// TIA Portal project "Practica_7_V14" (V14)
// Primer proyecto - practica experimental 7

(* hardware
DEVICE "S7-1200 station_1"  S7-1200 Station
   slot 0: "Rack_0"  Rack  V1.0
   slot 1: "PLC_1"  CPU 1214C DC/DC/DC  6ES7 214-1AG40-0XB0  V4.2
*)

// ===== PLC "PLC_1"  CPU 1214C DC/DC/DC =====

VAR_GLOBAL   // PLC tag table "Default tag table"
   "PM" AT %I0.0 : Bool;
   "PP" AT %I0.1 : Bool;
   "MOTOR" AT %Q0.0 : Bool;
   "APAGADO" AT %M0.1 : Bool;
   "ENCENDIDO" AT %M0.0 : Bool;
   "IL" AT %Q0.1 : Bool;
   "DP" AT %I0.2 : Bool;
   "CU" AT %M0.3 : Bool;
   "MEMORIA_RESET_CNT" AT %M0.2 : Bool;
END_VAR

// folder: System blocks/Program resources

DATA_BLOCK "CNT_UP"   // DB1
{ S7_Optimized_Access := 'TRUE' }
AUTHOR : Simatic
FAMILY : IEC
NAME : CNTR
VERSION : 1.0
// stored: InstanceOfName IEC_COUNTER
"IEC_COUNTER"
BEGIN
END_DATA_BLOCK

// folder: (top level)

ORGANIZATION_BLOCK "Main"   // OB1, LAD, ProgramCycle
TITLE = "Main Program Sweep (Cycle)"
{ S7_Optimized_Access := 'TRUE' }
VERSION : 0.1
   VAR_INPUT
      Initial_Call : Bool;   // Initial call of this OB
      Remanence : Bool;   // =True, if remanent data are available
   END_VAR
   VAR CONSTANT
      MAX_CNT : Int := 4;
   END_VAR
   VAR_TEMP   // added for the SCL form of the ladder/FBD networks
      _w1 : Bool;
   END_VAR
BEGIN

REGION Network 1
   // INICIALIZACION
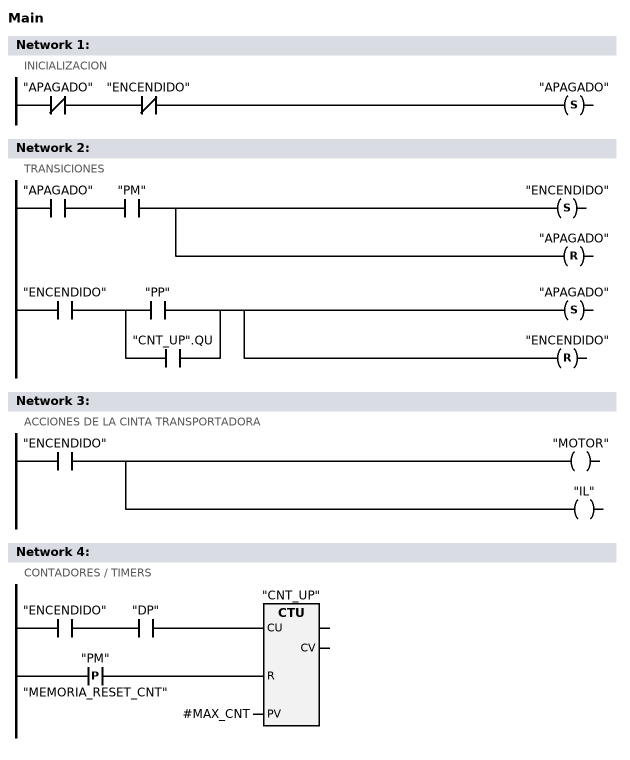
   RUNG wire#powerrail
      I_Contact( "APAGADO" )
      I_Contact( "ENCENDIDO" )
      S_Coil( "APAGADO" )
   END_RUNG
   // the same network as SCL:
   IF NOT "APAGADO" AND NOT "ENCENDIDO" THEN "APAGADO" := TRUE; END_IF;
END_REGION

REGION Network 2
   // TRANSICIONES
   RUNG wire#powerrail
      Contact( "APAGADO" )
      Contact( "PM" )
      wire#w1
      S_Coil( "ENCENDIDO" )
   END_RUNG
   RUNG wire#w1
      R_Coil( "APAGADO" )
   END_RUNG
   RUNG wire#powerrail
      Contact( "ENCENDIDO" )
      wire#w2
      Contact( "PP" )
      wire#w3
      S_Coil( "APAGADO" )
   END_RUNG
   RUNG wire#w2
      Contact( "CNT_UP".QU )
   END_RUNG wire#w3
   RUNG wire#w3
      R_Coil( "ENCENDIDO" )
   END_RUNG
   // the same network as SCL:
   IF "APAGADO" AND "PM" THEN
       "ENCENDIDO" := TRUE;
       "APAGADO" := FALSE;
   END_IF;
   IF "ENCENDIDO" AND ("PP" OR "CNT_UP".QU) THEN
       "APAGADO" := TRUE;
       "ENCENDIDO" := FALSE;
   END_IF;
END_REGION

REGION Network 3
   // ACCIONES DE LA CINTA TRANSPORTADORA
   RUNG wire#powerrail
      Contact( "ENCENDIDO" )
      wire#w1
      Coil( "MOTOR" )
   END_RUNG
   RUNG wire#w1
      Coil( "IL" )
   END_RUNG
   // the same network as SCL:
   "MOTOR" := "ENCENDIDO";
   "IL" := "ENCENDIDO";
END_REGION

REGION Network 4
   // CONTADORES / TIMERS
   #_w1 := "PM" AND NOT "MEMORIA_RESET_CNT";   // rising edge of "PM"
   "MEMORIA_RESET_CNT" := "PM";
   "CNT_UP".CTU(CU := "ENCENDIDO" AND "DP", R := #_w1, PV := #MAX_CNT);
END_REGION
END_ORGANIZATION_BLOCK